FUNCTION_BLOCK RegisterServiceHTTP (* Register Service using HTTP *)
  (* Standard: 61499-2; Description: Copyright (c) 2018 fortiss GmbH This program and the accompanying materials are made available under the terms of the Eclipse Public License 2.0 which is available at https://www.eclipse.org/legal/epl-2.0/ SPDX-License-Identifier: EPL-2.0 *)
  (* Version 1.0, 2018-09-21, Jose Cabral, fortiss GmbH *)
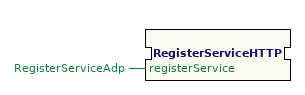
  SOCKETS
    registerService : RegisterServiceAdp; (* Register Service adapter *)
  END_SOCKETS
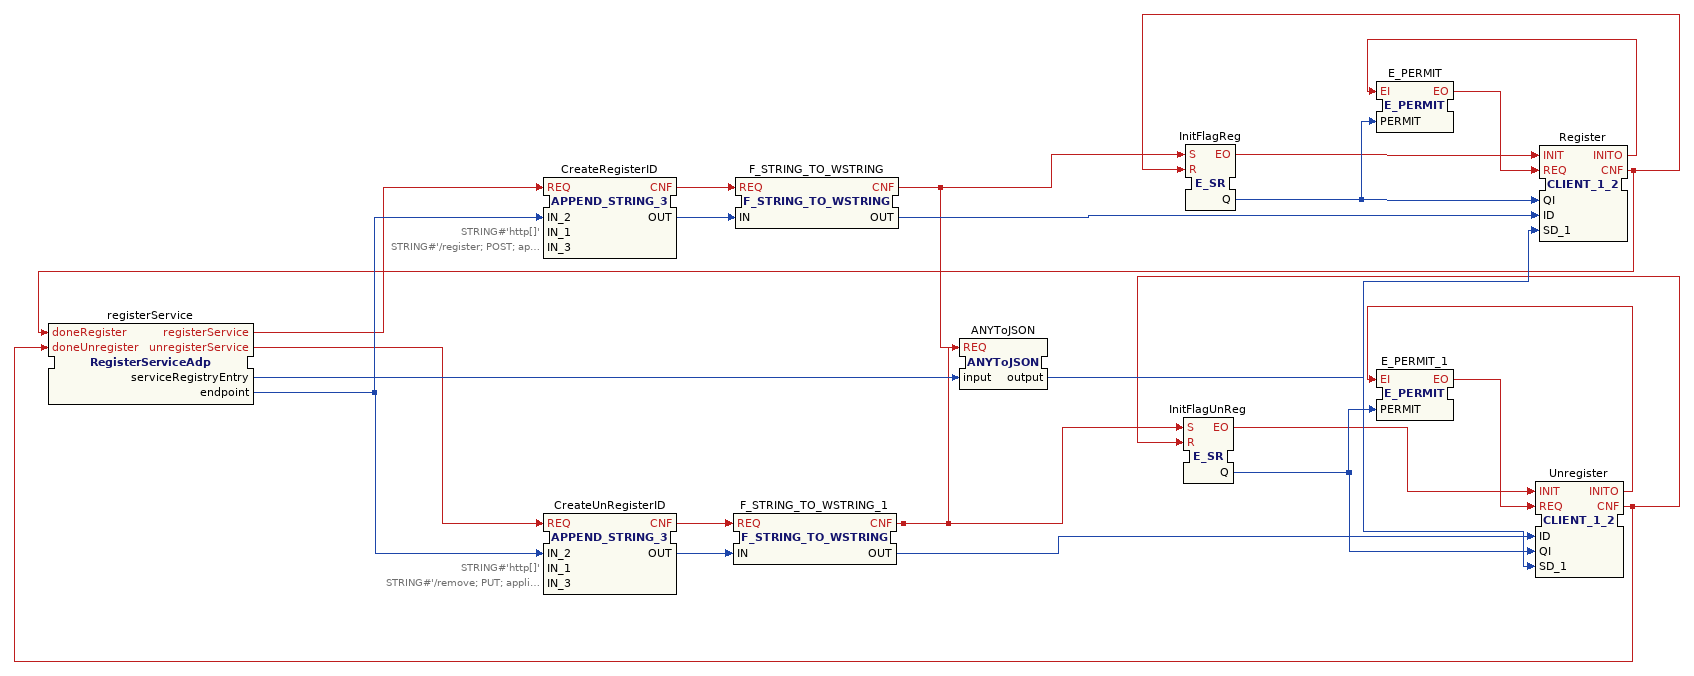
  FBS
    Register : CLIENT_1_2;
    Unregister : CLIENT_1_2;
    InitFlagReg : E_SR;
    E_PERMIT : E_PERMIT;
    CreateRegisterID : APPEND_STRING_3(IN_1 := STRING#'http[]', IN_3 := STRING#'/register; POST; application/json]');
    F_STRING_TO_WSTRING : F_STRING_TO_WSTRING;
    E_PERMIT_1 : E_PERMIT;
    InitFlagUnReg : E_SR;
    CreateUnRegisterID : APPEND_STRING_3(IN_1 := STRING#'http[]', IN_3 := STRING#'/remove; PUT; application/json]');
    F_STRING_TO_WSTRING_1 : F_STRING_TO_WSTRING;
    ANYToJSON : ANYToJSON;
  END_FBS
  EVENT_CONNECTIONS
    CreateRegisterID.CNF TO F_STRING_TO_WSTRING.REQ;
    F_STRING_TO_WSTRING.CNF TO InitFlagReg.S;
    CreateUnRegisterID.CNF TO F_STRING_TO_WSTRING_1.REQ;
    F_STRING_TO_WSTRING_1.CNF TO InitFlagUnReg.S;
    InitFlagUnReg.EO TO Unregister.INIT;
    Unregister.INITO TO E_PERMIT_1.EI;
    E_PERMIT_1.EO TO Unregister.REQ;
    Unregister.CNF TO InitFlagUnReg.R;
    InitFlagReg.EO TO Register.INIT;
    E_PERMIT.EO TO Register.REQ;
    Register.INITO TO E_PERMIT.EI;
    Register.CNF TO InitFlagReg.R;
    F_STRING_TO_WSTRING.CNF TO ANYToJSON.REQ;
    F_STRING_TO_WSTRING_1.CNF TO ANYToJSON.REQ;
    Register.CNF TO registerService.doneRegister;
    Unregister.CNF TO registerService.doneUnregister;
    registerService.registerService TO CreateRegisterID.REQ;
    registerService.unregisterService TO CreateUnRegisterID.REQ;
  END_CONNECTIONS
  DATA_CONNECTIONS
    InitFlagReg.Q TO E_PERMIT.PERMIT;
    CreateRegisterID.OUT TO F_STRING_TO_WSTRING.IN;
    CreateUnRegisterID.OUT TO F_STRING_TO_WSTRING_1.IN;
    F_STRING_TO_WSTRING_1.OUT TO Unregister.ID;
    InitFlagUnReg.Q TO Unregister.QI;
    InitFlagUnReg.Q TO E_PERMIT_1.PERMIT;
    InitFlagReg.Q TO Register.QI;
    F_STRING_TO_WSTRING.OUT TO Register.ID;
    ANYToJSON.output TO Register.SD_1;
    ANYToJSON.output TO Unregister.SD_1;
    registerService.serviceRegistryEntry TO ANYToJSON.input;
    registerService.endpoint TO CreateRegisterID.IN_2;
    registerService.endpoint TO CreateUnRegisterID.IN_2;
  END_CONNECTIONS
END_FUNCTION_BLOCK
